(* IEC 61131-3 sources: Industry-PLC-LLM/data/PLCBEAD_repo/PLCBEAD_PLCEmbed-main/PLC-BEAD/Source/GEB/BCDC_TO_INT, 1 file *)

(* ---- BCDC_TO_INT.ST ---- *)
FUNCTION _BYTE_TO_INT:INT
	VAR_INPUT
		IN :	BYTE;
	END_VAR

	_BYTE_TO_INT := USINT_TO_INT(BYTE_TO_USINT(IN));

END_FUNCTION

FUNCTION BCDC_TO_INT:INT
	VAR_INPUT
		IN :	BYTE;
	END_VAR

	BCDC_TO_INT := _BYTE_TO_INT(IN AND BYTE#16#0F) + (_BYTE_TO_INT(SHR(IN,4)) * 10);
END_FUNCTION

PROGRAM program0
  VAR
    LocalVar0 : BYTE;
    LocalOUT  : INT;
  END_VAR

  LocalOUT := BCDC_TO_INT(LocalVar0);
END_PROGRAM
